ABB RobotStudio station: Celda.rsstn

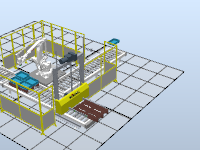
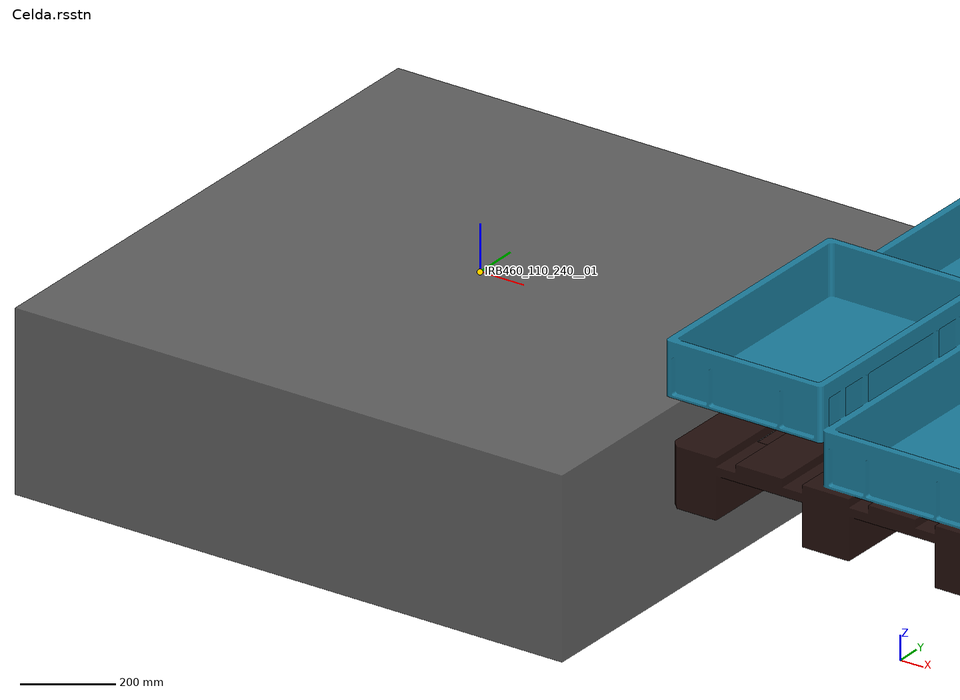
[picture v1: parts stored in the station drawn from their meshes, with robot base, taught points and paths (robot models come from the ABB library and are not in the file)]
Station Celda (saved by RobotStudio 21.2.9526.0)
Controller Controller2, task T_ROB1: task frame (RAPID world) sits at (0, 0, 435) mm in the station
Controller Controller2
  mechanical unit ROB_1: IRB460_110_240__01, 6 joints, base frame (0, 0, 0) mm
Layout (positions relative to the parent item):
  - IRB460_110_240__01 [mechanism, from Robots\IRB460_110_240__02.rslib] at (0, 0, 435) mm; joint values [-0.0882, -0.0322, 0.3232, -0.0882] (rad or m)
  - DispenserPallet [part] at (1350, 4000, 435) mm, rotated rx 90 ry 0 rz 180 deg, size 1784 x 3045 x 1697.6 mm
  - 950_4800_h2 [part, from Equipment\Conveyor 950 4800 h2.rslib] at (-4200, 850, 0) mm
  - 950_4800_h2_2 [part, from Equipment\Conveyor 950 4800 h2.rslib] at (900, 4000, 0) mm, rotated rx 0 ry 0 rz -90 deg
  - Part_2 [part] at (-700, -700, 0) mm, size 1400 x 1400 x 435 mm
  - Plastic crate 600x400x120_2 [part] at (-4105.7, 1135.15, 1018.04) mm, size 600 x 400 x 140 mm
  - Euro Pallet [graphiccomponentgroup] at (3161.81, 690.63, 699.77) mm, rotated rx 0 ry 0 rz 90 deg
    - Body 1 [part] at (2624.7, 1387.85, 0) mm, size 1200 x 800 x 144 mm
  - Fence_2500 [graphiccomponentgroup, from Equipment\Fence_2500.rslib] at (-2079.28, 2740, 0) mm, rotated rx 0 ry 0 rz -90 deg
    - Body 1 [part, from Equipment\Fence_2500.rslib]
    - Body 2 [part, from Equipment\Fence_2500.rslib]
  - Fence_740 [graphiccomponentgroup, from Equipment\Fence_740.rslib] at (-2100, 2000, 0) mm
    - Body 1 [part, from Equipment\Fence_740.rslib]
    - Body 2 [part, from Equipment\Fence_740.rslib]
  - 950_4000_h2_2 [part, from Equipment\Conveyor 950 4000 h2.rslib] at (900, -1050, 0) mm, rotated rx 0 ry 0 rz -90 deg
  - Fence_2502 [graphiccomponentgroup, from Equipment\Fence_2500.rslib] at (3000, -2235.69, 0) mm
    - Body 1 [part, from Equipment\Fence_2500.rslib]
    - Body 2 [part, from Equipment\Fence_2500.rslib]
  - Fence_2503 [graphiccomponentgroup, from Equipment\Fence_2500.rslib] at (3000, 238.8, 0) mm
    - Body 1 [part, from Equipment\Fence_2500.rslib]
    - Body 2 [part, from Equipment\Fence_2500.rslib]
  - Gate [graphiccomponentgroup, from Equipment\Fence_Gate.rslib] at (-2100, 728.56, 0) mm, rotated rx 0 ry 0 rz 180 deg
    - Body 1 [part, from Equipment\Fence_Gate.rslib]
    - Body 2 [part, from Equipment\Fence_Gate.rslib]
    - Body 3 [part, from Equipment\Fence_Gate.rslib]
  - Fence_740_2 [graphiccomponentgroup, from Equipment\Fence_740.rslib] at (3000, 2740, 0) mm, rotated rx 0 ry 0 rz 90 deg
    - Body 1 [part, from Equipment\Fence_740.rslib]
    - Body 2 [part, from Equipment\Fence_740.rslib]
  - Fence_740_3 [graphiccomponentgroup, from Equipment\Fence_740.rslib] at (-2100, -1490.03, 0) mm
    - Body 1 [part, from Equipment\Fence_740.rslib]
    - Body 2 [part, from Equipment\Fence_740.rslib]
  - Fence_740_4 [graphiccomponentgroup, from Equipment\Fence_740.rslib] at (-2153.49, -2200, 0) mm, rotated rx 0 ry 0 rz -90 deg
    - Body 1 [part, from Equipment\Fence_740.rslib]
    - Body 2 [part, from Equipment\Fence_740.rslib]
  - Fence_740_8 [graphiccomponentgroup, from Equipment\Fence_740.rslib] at (-1386.41, -2200, 0) mm, rotated rx 0 ry 0 rz -90 deg
    - Body 1 [part, from Equipment\Fence_740.rslib]
    - Body 2 [part, from Equipment\Fence_740.rslib]
  - Fence_740_9 [graphiccomponentgroup, from Equipment\Fence_740.rslib] at (-657.15, -2200, 0) mm, rotated rx 0 ry 0 rz -90 deg
    - Body 1 [part, from Equipment\Fence_740.rslib]
    - Body 2 [part, from Equipment\Fence_740.rslib]
  - Fence_740_10 [graphiccomponentgroup, from Equipment\Fence_740.rslib] at (82.68, -2200, 0) mm, rotated rx 0 ry 0 rz -90 deg
    - Body 1 [part, from Equipment\Fence_740.rslib]
    - Body 2 [part, from Equipment\Fence_740.rslib]
  - Fence_740_11 [graphiccomponentgroup, from Equipment\Fence_740.rslib] at (-2100, -2267.47, 0) mm
    - Body 1 [part, from Equipment\Fence_740.rslib]
    - Body 2 [part, from Equipment\Fence_740.rslib]
  - Fence_740_12 [graphiccomponentgroup, from Equipment\Fence_740.rslib] at (3000, -2297.98, 0) mm, rotated rx 0 ry 0 rz 90 deg
    - Body 1 [part, from Equipment\Fence_740.rslib]
    - Body 2 [part, from Equipment\Fence_740.rslib]
  - Euro Pallet_2 [graphiccomponentgroup] at (3411.22, -3314.71, 435) mm, rotated rx 0 ry 0 rz 90 deg
    - Body 1 [part] at (2624.7, 1644.3, 0) mm, size 1200 x 800 x 144 mm
  - Plastic crate 600x400x120_3 [part] at (1353.48, -686.24, 677) mm, rotated rx 0 ry 0 rz 90 deg, size 600 x 400 x 140 mm
  - Plastic crate 600x400x120_7 [part] at (1754.81, -85.7, 577) mm, rotated rx 0 ry 0 rz 90 deg, size 600 x 400 x 140 mm
  - Plastic crate 600x400x120_8 [part] at (1353.78, -84.84, 577) mm, rotated rx 0 ry 0 rz 90 deg, size 600 x 400 x 140 mm
  - Plastic crate 600x400x120_9 [part] at (1754.81, -686.44, 577) mm, rotated rx 0 ry 0 rz 90 deg, size 600 x 400 x 140 mm
  - Gripper [mechanism] at (1415.95, -125.24, 1544.98) mm, rotated rx 180 ry 0 rz 180 deg
      TCP Gripper at (1415.95, -125.24, 1544.98) mm, rotated rx -180 ry 0 rz 180 deg
      links: gripper_2
  - SmartComponent_1 [smart component]
Targets, tools, work objects and paths stored in the station, written as RAPID:
! task T_ROB1
MODULE CalibData
  PERS tooldata Gripper:=[TRUE,[[1415.95,-125.238,1544.984],[0,0,1,0]],[45,[41.46,0.078,112.5],[1,0,0,0],7047,6515,11100]];
ENDMODULE

! task T_ROB1
MODULE Module1
  CONST robtarget Target_10:=[[-0.000025482,-250.476405368,-434.999924838],[1,0,0,0],[-1,0,-1,0],[9E+09,9E+09,9E+09,9E+09,9E+09,9E+09]];
  PROC Path_10()
  ENDPROC
ENDMODULE

